//Use for testing purposes to set the attenuator status to a good state
FUNCTION F_SetGoodAttStatus : UINT
VAR_INPUT
    xStatus : UINT;
END_VAR
VAR
END_VAR

xStatus.0 := 1;
xStatus.3 := 1;
xStatus.4 := 1;

END_FUNCTION

(* stored: Version 1.1.0.1
   POU F_SetGoodAttStatus: Id {e6cd67bb-2bd9-4b3d-9199-950e5913b39f}, SpecialFunc None *)
